Universal Robots PolyScope program: verticalMove.urp

Program verticalMove (installation=default directory=/ursim/programs createdIn=5.19.0 lastSavedIn=5.19.0 robotSerialNumber=20195599999)
Calibrated DH parameters: a=[0, -0.425, -0.3922, 0, 0, 0]; d=[0.1625, 0, 0, 0.1333, 0.0997, 0.0996]; alpha=[1.570796, 0, 0, 1.570796, -1.570796, 0]; deltaTheta=[0, 0, 0, 0, 0, 0]
InitVariablesNode
Robot Program (runOnlyOnce=false)
  Script: reset_world_model()
  Script: add_frame("vTCP", p[0.286,0,0.690,0,1.57,0],"world")
  Script: thread move_vTCPThread(): move_vTCP() end
  Script: movej("vTCP")
  Script: frame_tracking_enable("world")
  Script: thrd = run move_vTCPThread()
  Loop Forever
    Script: movel(struct(pose=p[0,0.2,0,0,0,0],frame ="vTCP"), v= 0.1)
    Script: movel(struct(pose=p[0,-0.2,0,0,0,0],frame ="vTCP"), v=0.1)
SubProgram move_vTCP (keepSynchronizedWithDisk=false)
  Script: A=2
  Script: p=0
  Script: w=0.2
  Loop Forever
    Script: p = p + w*(2*3.1416/500)
    Script: move_frame("vTCP", p[0.286,0,0.69+0.3*sin(p),0,1.57,0],"world")
    Script: sync()
